PROGRAM Main5
VAR
END_VAR

END_PROGRAM

(* stored: Version 1.1.0.1, ProductVersion 3.1.4024.11
   POU Main5: Id {686a13c3-5a9c-4afd-94a3-f410a29c8d2f}, SpecialFunc None *)
